TYPE ST_TechnosoftMotionError :
STRUCT
    bit0_EtherCATCommunicationError: BIT; //EtherCAT communication error
    bit1_ShortCircuit: BIT; //Short circuit
    bit2_InvalidSetupData: BIT; //Invalid setup data
    bit3_ControlError: BIT; //Position or speed error
    bit4_CommunicationError: BIT; //Communication error
    bit5_FeedbackError: BIT; //Feedback error
    bit6_PositiveLimitSwitchActive: BIT; //Positive limit active
    bit7_NegativeLimitSwitchActive: BIT; //Negative limit active
    bit8_OverCurrent: BIT; //Over current
    bit9_I2TProtection: BIT; //I2T protection active
    bit10_MotorOverTemperature: BIT; //Motor over temperature
    bit11_DriveOverTemperature: BIT; //Drive over temperature
    bit12_OverVoltage: BIT; //Over voltage
    bit13_UnderVoltage: BIT; //Under voltage
    bit14_CommandError: BIT; //Command error
    bit15_STOActive: BIT; //Enabled or STO disabled
END_STRUCT
END_TYPE

(* stored: Version 1.1.0.1
   DUT ST_TechnosoftMotionError: Id {fc262979-66dd-0743-2a0b-48ac6294268e} *)
